FUNCTION AnalogScaler : LREAL
VAR_INPUT
	input : LREAL;
	rawLow : LREAL;
	rawHigh : LREAL;
	processLow : LREAL;
	processHigh : LREAL;
END_VAR

AnalogScaler := (processHigh - processLow)
	* (input - rawLow)
	/ (rawHigh - rawLow)
	+ processLow;

END_FUNCTION

(* stored: Version 1.1.0.1, ProductVersion 3.1.4024.12
   POU AnalogScaler: Id {bd8f0ae4-3515-0ad5-3888-f8451597a613}, SpecialFunc None *)
